{attribute 'GeneratedUsingTerminal: EL3751-0000-0020'}
{attribute addProperty BoxType "EL3751-0000-0020"}
{attribute addProperty Id "LowUDINT4HiUDINT4"}
{attribute addProperty CRC "48284104"}
{attribute addProperty Size "8"}
TYPE StartTimeNextLatch_02E0C1C8 :
STRUCT
	{attribute addProperty Name "Low"}
	Low : UDINT;
	{attribute addProperty Name "Hi"}
	Hi : UDINT;
END_STRUCT
END_TYPE

(* stored: Version 1.2.0.0, ProductVersion 3.1.4024.9
   DUT StartTimeNextLatch_02E0C1C8: Id {c952b43b-a214-486e-8b3e-c86da1d04c3d} *)
